FUNCTION_BLOCK FB_Component2 EXTENDS FB_BaseComponent IMPLEMENTS ITF_Component2, ITF_Component2_HMI_Connector
VAR
END_VAR

END_FUNCTION_BLOCK

(* stored: Version 1.1.0.1
   POU FB_Component2: Id {d0df42df-9590-0ba4-291d-f5acb6da50c9}, SpecialFunc None *)
